// TIA Portal V18 export
// export: Created 2026-03-12T16:03:53.211165Z, ExportSetting WithDefaults, DisplayName Totally Integrated Automation Portal, DisplayVersion V18 Update 5, DisplayName TIA Portal Openness, DisplayVersion V18 Update 5, DisplayName TIA Portal Version Control Interface, DisplayVersion V18, DisplayName SINAMICS Startdrive Advanced, DisplayVersion V18, DisplayName SINAMICS Startdrive G130, G150, S120, S150, SINAMICS MV, S210, DisplayVersion V18, DisplayName SINAMICS Startdrive G110M, G120, G120C, G120D, G120P, G115D, DisplayVersion V18, DisplayName STEP 7 Professional, DisplayVersion V18 Update 5, DisplayName STEP 7 Safety, DisplayVersion V18, DisplayName WinCC Professional, DisplayVersion V18 Update 5
TagTable "TAG_ELE_GORDURA"
  DB GLOBAL_ELEVATÓRIA_DE_GORDURA_COMANDO_BOMBA_SDG_RESET_HORIMETRO : Bool  (PLC tag "DB GLOBAL".ELEVATORIA_DE_GORDURA.COMANDO.BOMBA_SDG.RESET_HORIMETRO, HMI_Connection_6, 1 s)
  DB GLOBAL_ELEVATÓRIA_DE_GORDURA_BOMBA_SDG_HORIMETRO : UInt  (PLC tag "DB GLOBAL".ELEVATORIA_DE_GORDURA.BOMBA_SDG.HORIMETRO, HMI_Connection_6, 1 s)
  DB GLOBAL_ELEVATORIA_DE_GORDURA_BOMBA_BH-01A_REF_TORQUE : Real  (PLC tag "DB GLOBAL".ELEVATORIA_DE_GORDURA.BOMBA_BH-01A.REF_TORQUE, HMI_Connection_6, 1 s)
  DB GLOBAL_ELEVATÓRIA_DE_GORDURA_COMANDO_CONJUNTO_BOMBA_BH-01A_&_BH-01B_MANUTENCAO_PRINCIPAL : Bool  (PLC tag "DB GLOBAL".ELEVATORIA_DE_GORDURA.COMANDO.CONJUNTO_BOMBA_BH-01A_&_BH-01B.MANUTENCAO_PRINCIPAL, HMI_Connection_6, 1 s)
  DB GLOBAL_ELEVATORIA_DE_GORDURA_BOMBA_BH-01B_REF_POTENCIA : Real  (PLC tag "DB GLOBAL".ELEVATORIA_DE_GORDURA.BOMBA_BH-01B.REF_POTENCIA, HMI_Connection_6, 1 s)
  DB GLOBAL_ELEVATORIA_DE_GORDURA_BOMBA_BH-01A_CADASTRO_MAX_LEITURA : Int  (PLC tag "DB GLOBAL".ELEVATORIA_DE_GORDURA.BOMBA_BH-01A.CADASTRO_MAX_LEITURA, HMI_Connection_6, 1 s)
  DB GLOBAL_ELEVATORIA_DE_GORDURA_BOMBA_BH-01A_REF_VELOCIDADE : Real  (PLC tag "DB GLOBAL".ELEVATORIA_DE_GORDURA.BOMBA_BH-01A.REF_VELOCIDADE, HMI_Connection_6, 1 s)
  DB GLOBAL_ELEVATÓRIA_DE_GORDURA_COMANDO_CONJUNTO_BOMBA_BH-01A_&_BH-01B_RESET_HORIMETRO_PRINCIPAL : Bool  (PLC tag "DB GLOBAL".ELEVATORIA_DE_GORDURA.COMANDO.CONJUNTO_BOMBA_BH-01A_&_BH-01B.RESET_HORIMETRO_PRINCIPAL, HMI_Connection_6, 1 s)
  DB GLOBAL_ELEVATÓRIA_DE_GORDURA_COMANDO_BOMBA_SDG_LIGA : Bool  (PLC tag "DB GLOBAL".ELEVATORIA_DE_GORDURA.COMANDO.BOMBA_SDG.LIGA, HMI_Connection_6, 1 s)
  DB GLOBAL_ELEVATÓRIA_DE_GORDURA_SENSORES_SENSOR_HIDROSTÁTICO_LT-04_CADASTRO_MAX : Int  (PLC tag "DB GLOBAL".ELEVATORIA_DE_GORDURA.SENSORES.SENSOR_HIDROSTÁTICO_LT-04.CADASTRO_MAX, HMI_Connection_6, 1 s)
  DB GLOBAL_ELEVATÓRIA_DE_GORDURA_SENSORES_SENSOR_HIDROSTÁTICO_LT-04_CADASTRO_LEITURA_MUITO_BAIXA : Real  (PLC tag "DB GLOBAL".ELEVATORIA_DE_GORDURA.SENSORES.SENSOR_HIDROSTÁTICO_LT-04.CADASTRO_LEITURA_MUITO_BAIXA, HMI_Connection_6, 1 s)
  DB GLOBAL_ELEVATÓRIA_DE_GORDURA_COMANDO_CONJUNTO_BOMBA_BH-01A_&_BH-01B_MANUTENCAO_RESERVA : Bool  (PLC tag "DB GLOBAL".ELEVATORIA_DE_GORDURA.COMANDO.CONJUNTO_BOMBA_BH-01A_&_BH-01B.MANUTENCAO_RESERVA, HMI_Connection_6, 1 s)
  DB GLOBAL_ELEVATÓRIA_DE_GORDURA_SENSORES_SENSOR_HIDROSTÁTICO_LT-04_CADASTRO_LEITURA_MUITO_ALTA : Real  (PLC tag "DB GLOBAL".ELEVATORIA_DE_GORDURA.SENSORES.SENSOR_HIDROSTÁTICO_LT-04.CADASTRO_LEITURA_MUITO_ALTA, HMI_Connection_6, 1 s)
  DB GLOBAL_ELEVATÓRIA_DE_GORDURA_BOMBA_SDG_STATUS_MOTOR : Byte  (PLC tag "DB GLOBAL".ELEVATORIA_DE_GORDURA.BOMBA_SDG.STATUS_MOTOR, HMI_Connection_6, 1 s)
  DB GLOBAL_ELEVATORIA_DE_GORDURA_BOMBA_BH-01A_VELOCIDADE : Int  (PLC tag "DB GLOBAL".ELEVATORIA_DE_GORDURA.BOMBA_BH-01A.VELOCIDADE, HMI_Connection_6, 1 s)
  DB GLOBAL_ELEVATORIA_DE_GORDURA_BOMBA_BH-01B_OPERACAO_MOTOR : Byte  (PLC tag "DB GLOBAL".ELEVATORIA_DE_GORDURA.BOMBA_BH-01B.OPERACAO_MOTOR, HMI_Connection_6, 1 s)
  DB GLOBAL_ELEVATÓRIA_DE_GORDURA_COMANDO_BOMBA_SDG_RESET_FALHA : Bool  (PLC tag "DB GLOBAL".ELEVATORIA_DE_GORDURA.COMANDO.BOMBA_SDG.RESET_FALHA, HMI_Connection_6, 1 s)
  DB GLOBAL_ELEVATORIA_DE_GORDURA_BOMBA_BH-01A_REF_POTENCIA : Real  (PLC tag "DB GLOBAL".ELEVATORIA_DE_GORDURA.BOMBA_BH-01A.REF_POTENCIA, HMI_Connection_6, 1 s)
  DB GLOBAL_ELEVATÓRIA_DE_GORDURA_BOMBA_SDG_OPERACAO_MOTOR : Byte  (PLC tag "DB GLOBAL".ELEVATORIA_DE_GORDURA.BOMBA_SDG.OPERACAO_MOTOR, HMI_Connection_6, 1 s)
  DB GLOBAL_ELEVATÓRIA_DE_GORDURA_SENSORES_SENSOR_HIDROSTÁTICO_LT-04_CADASTRO_LEITURA_BAIXA : Real  (PLC tag "DB GLOBAL".ELEVATORIA_DE_GORDURA.SENSORES.SENSOR_HIDROSTÁTICO_LT-04.CADASTRO_LEITURA_BAIXA, HMI_Connection_6, 1 s)
  DB GLOBAL_ELEVATÓRIA_DE_GORDURA_COMANDO_BOMBA_SDG_MANUTENCAO : Bool  (PLC tag "DB GLOBAL".ELEVATORIA_DE_GORDURA.COMANDO.BOMBA_SDG.MANUTENCAO, HMI_Connection_6, 1 s)
  DB GLOBAL_ELEVATORIA_DE_GORDURA_BOMBA_BH-01A_REF_CORRENTE : Real  (PLC tag "DB GLOBAL".ELEVATORIA_DE_GORDURA.BOMBA_BH-01A.REF_CORRENTE, HMI_Connection_6, 1 s)
  DB GLOBAL_ELEVATÓRIA_DE_GORDURA_BOMBA_BH-01B_STATUS_MOTOR : Byte  (PLC tag "DB GLOBAL".ELEVATORIA_DE_GORDURA.BOMBA_BH-01B.STATUS_MOTOR, HMI_Connection_6, 1 s)
  DB GLOBAL_ELEVATORIA_DE_GORDURA_BOMBA_BH-01B_CADASTRO_MAX_LEITURA : Int  (PLC tag "DB GLOBAL".ELEVATORIA_DE_GORDURA.BOMBA_BH-01B.CADASTRO_MAX_LEITURA, HMI_Connection_6, 1 s)
  DB GLOBAL_ELEVATÓRIA_DE_GORDURA_BOMBA_BH-01A_HORIMETRO : UInt  (PLC tag "DB GLOBAL".ELEVATORIA_DE_GORDURA.BOMBA_BH-01A.HORIMETRO, HMI_Connection_6, 1 s)
  DB GLOBAL_ELEVATÓRIA_DE_GORDURA_COMANDO_CONJUNTO_BOMBA_BH-01A_&_BH-01B_HABILITA : Int  (PLC tag "DB GLOBAL".ELEVATORIA_DE_GORDURA.COMANDO.CONJUNTO_BOMBA_BH-01A_&_BH-01B.HABILITA, HMI_Connection_6, 1 s)
  DB GLOBAL_ELEVATÓRIA_DE_GORDURA_BOMBA_BH-01A_OPERACAO_MOTOR : Byte  (PLC tag "DB GLOBAL".ELEVATORIA_DE_GORDURA.BOMBA_BH-01A.OPERACAO_MOTOR, HMI_Connection_6, 1 s)
  DB GLOBAL_ELEVATÓRIA_DE_GORDURA_COMANDO_CONJUNTO_BOMBA_BH-01A_&_BH-01B_MODO_OPERACAO : Bool  (PLC tag "DB GLOBAL".ELEVATORIA_DE_GORDURA.COMANDO.CONJUNTO_BOMBA_BH-01A_&_BH-01B.MODO_OPERACAO, HMI_Connection_6, 1 s)
  DB GLOBAL_ELEVATORIA_DE_GORDURA_BOMBA_BH-01B_CADASTRO_MIN_LEITURA : Int  (PLC tag "DB GLOBAL".ELEVATORIA_DE_GORDURA.BOMBA_BH-01B.CADASTRO_MIN_LEITURA, HMI_Connection_6, 1 s)
  DB GLOBAL_ELEVATÓRIA_DE_GORDURA_COMANDO_CONJUNTO_BOMBA_BH-01A_&_BH-01B_RESET_FALHA_RESERVA : Bool  (PLC tag "DB GLOBAL".ELEVATORIA_DE_GORDURA.COMANDO.CONJUNTO_BOMBA_BH-01A_&_BH-01B.RESET_FALHA_RESERVA, HMI_Connection_6, 1 s)
  DB GLOBAL_ELEVATORIA_DE_GORDURA_BOMBA_BH-01B_REF_CORRENTE : Real  (PLC tag "DB GLOBAL".ELEVATORIA_DE_GORDURA.BOMBA_BH-01B.REF_CORRENTE, HMI_Connection_6, 1 s)
  DB GLOBAL_ELEVATORIA_DE_GORDURA_BOMBA_BH-01A_SETPOINT_MANUAL : Int  (PLC tag "DB GLOBAL".ELEVATORIA_DE_GORDURA.BOMBA_BH-01A.SETPOINT_MANUAL, HMI_Connection_6, 1 s)
  DB GLOBAL_ELEVATORIA_DE_GORDURA_BOMBA_BH-01B_VELOCIDADE : Int  (PLC tag "DB GLOBAL".ELEVATORIA_DE_GORDURA.BOMBA_BH-01B.VELOCIDADE, HMI_Connection_6, 1 s)
  DB GLOBAL_ELEVATÓRIA_DE_GORDURA_BOMBA_BH-01B_HORIMETRO : UInt  (PLC tag "DB GLOBAL".ELEVATORIA_DE_GORDURA.BOMBA_BH-01B.HORIMETRO, HMI_Connection_6, 1 s)
  DB GLOBAL_ELEVATÓRIA_DE_GORDURA_COMANDO_CONJUNTO_BOMBA_BH-01A_&_BH-01B_LIGA : Bool  (PLC tag "DB GLOBAL".ELEVATORIA_DE_GORDURA.COMANDO.CONJUNTO_BOMBA_BH-01A_&_BH-01B.LIGA, HMI_Connection_6, 1 s)
  DB GLOBAL_ELEVATORIA_DE_GORDURA_BOMBA_BH-01A_CADASTRO_MIN_LEITURA : Int  (PLC tag "DB GLOBAL".ELEVATORIA_DE_GORDURA.BOMBA_BH-01A.CADASTRO_MIN_LEITURA, HMI_Connection_6, 1 s)
  DB GLOBAL_ELEVATORIA_DE_GORDURA_BOMBA_BH-01B_REF_TORQUE : Real  (PLC tag "DB GLOBAL".ELEVATORIA_DE_GORDURA.BOMBA_BH-01B.REF_TORQUE, HMI_Connection_6, 1 s)
  DB GLOBAL_ELEVATÓRIA_DE_GORDURA_SENSORES_SENSOR_HIDROSTÁTICO_LT-04_CADASTRO_LEITURA_ALTA : Real  (PLC tag "DB GLOBAL".ELEVATORIA_DE_GORDURA.SENSORES.SENSOR_HIDROSTÁTICO_LT-04.CADASTRO_LEITURA_ALTA, HMI_Connection_6, 1 s)
  DB GLOBAL_ELEVATÓRIA_DE_GORDURA_COMANDO_CONJUNTO_BOMBA_BH-01A_&_BH-01B_RESET_FALHA_PRINCIPAL : Bool  (PLC tag "DB GLOBAL".ELEVATORIA_DE_GORDURA.COMANDO.CONJUNTO_BOMBA_BH-01A_&_BH-01B.RESET_FALHA_PRINCIPAL, HMI_Connection_6, 1 s)
  DB GLOBAL_ELEVATORIA_DE_GORDURA_COMANDO_CONJUNTO_BOMBA_BH-01A_&_BH-01B_INTERTRAVAMENTO_LIGA : Bool  (PLC tag "DB GLOBAL".ELEVATORIA_DE_GORDURA.COMANDO.CONJUNTO_BOMBA_BH-01A_&_BH-01B.INTERTRAVAMENTO_LIGA, HMI_Connection_6, 1 s)
  DB GLOBAL_ELEVATORIA_DE_GORDURA_BOMBA_BH-01B_SETPOINT_MANUAL : Int  (PLC tag "DB GLOBAL".ELEVATORIA_DE_GORDURA.BOMBA_BH-01B.SETPOINT_MANUAL, HMI_Connection_6, 1 s)
  DB GLOBAL_ELEVATORIA_DE_GORDURA_COMANDO_BOMBA_SDG_INTERTRAVAMENTO_LIGA : Bool  (PLC tag "DB GLOBAL".ELEVATORIA_DE_GORDURA.COMANDO.BOMBA_SDG.INTERTRAVAMENTO_LIGA, HMI_Connection_6, 1 s)
  DB GLOBAL_ELEVATÓRIA_DE_GORDURA_BOMBA_BH-01A_STATUS_MOTOR : Byte  (PLC tag "DB GLOBAL".ELEVATORIA_DE_GORDURA.BOMBA_BH-01A.STATUS_MOTOR, HMI_Connection_6, 1 s)
  DB GLOBAL_ELEVATÓRIA_DE_GORDURA_SENSORES_SENSOR_HIDROSTÁTICO_LT-04_STATUS_SENSOR : Real  (PLC tag "DB GLOBAL".ELEVATORIA_DE_GORDURA.SENSORES.SENSOR_HIDROSTÁTICO_LT-04.STATUS_SENSOR, HMI_Connection_6, 1 s)
  DB GLOBAL_ELEVATÓRIA_DE_GORDURA_SENSORES_SENSOR_HIDROSTÁTICO_LT-04_MANUTENÇÃO : Bool  (PLC tag "DB GLOBAL".ELEVATORIA_DE_GORDURA.SENSORES.SENSOR_HIDROSTÁTICO_LT-04.MANUTENCAO, HMI_Connection_6, 1 s)
  DB GLOBAL_ELEVATÓRIA_DE_GORDURA_COMANDO_BOMBA_SDG_MODO_OPERACAO : Bool  (PLC tag "DB GLOBAL".ELEVATORIA_DE_GORDURA.COMANDO.BOMBA_SDG.MODO_OPERACAO, HMI_Connection_6, 1 s)
  DB GLOBAL_ELEVATÓRIA_DE_GORDURA_SENSORES_SENSOR_HIDROSTÁTICO_LT-04_CADASTRO_MIN : Int  (PLC tag "DB GLOBAL".ELEVATORIA_DE_GORDURA.SENSORES.SENSOR_HIDROSTÁTICO_LT-04.CADASTRO_MIN, HMI_Connection_6, 1 s)
  DB GLOBAL_ELEVATORIA_DE_GORDURA_BOMBA_BH-01B_REF_VELOCIDADE : Real  (PLC tag "DB GLOBAL".ELEVATORIA_DE_GORDURA.BOMBA_BH-01B.REF_VELOCIDADE, HMI_Connection_6, 1 s)
  DB GLOBAL_ELEVATÓRIA_DE_GORDURA_COMANDO_CONJUNTO_BOMBA_BH-01A_&_BH-01B_RESET_HORIMETRO_RESERVA : Bool  (PLC tag "DB GLOBAL".ELEVATORIA_DE_GORDURA.COMANDO.CONJUNTO_BOMBA_BH-01A_&_BH-01B.RESET_HORIMETRO_RESERVA, HMI_Connection_6, 1 s)
  DB GLOBAL_ELEVATÓRIA_DE_GORDURA_SENSORES_SENSOR_HIDROSTÁTICO_LT-04_AMOSTRA_SENSOR : Int  (PLC tag "DB GLOBAL".ELEVATORIA_DE_GORDURA.SENSORES.SENSOR_HIDROSTÁTICO_LT-04.AMOSTRA_SENSOR, HMI_Connection_6, 1 s)
